Staubli VAL3: getTool.pgx

public program getTool(num& x_nTool)
begin
end
